{attribute 'GeneratedUsingTerminal: EK1960-2600-0019'}
{attribute addProperty BoxType "EK1960-2600-0019"}
{attribute addProperty Id "FSOEAT %Q*FSOE_CEFF8C5656"}
{attribute addProperty CRC "2012837978"}
{attribute addProperty Size "56"}
TYPE FSoE_Outputs_77F9785A :
STRUCT
	{attribute addProperty Name "FSOE"}
	FSOE AT %Q* : FSOE_CEFF8C56;
END_STRUCT
END_TYPE

(* stored: Version 1.2.0.0, ProductVersion 3.1.4024.9
   DUT FSoE_Outputs_77F9785A: Id {a2d5bf61-9fe0-46a9-8fe5-a9b9bc3bdf86} *)
